{attribute 'pack_mode' := '1'}
TYPE ST_OutputArgInfoAndData :
STRUCT
	nNumberOfOutputArguments: UDINT; // determined amount of output parameters
	nReserved: ARRAY[1..4] OF BYTE; // Reserved padding
	stOutputArgInfo: ARRAY[1..1] OF ST_UAMethodArgInfo; // number of output parameters - M_Mul has 1 output parameter 
	pro: DINT;
END_STRUCT
END_TYPE

(* stored: Version 1.1.0.1, ProductVersion 3.1.4024.10
   DUT ST_OutputArgInfoAndData: Id {aa411b33-0ffd-48f8-ad37-0dd63243bc1d} *)
